INTERFACE I_Level EXTENDS I_Component

METHOD PUBLIC M_Attach : BOOL
VAR_INPUT
	iObject: 	I_Component;
END_VAR
END_METHOD

METHOD PUBLIC M_Detach : BOOL
VAR_INPUT
	iObject: 	I_Component;
END_VAR
END_METHOD

{attribute 'OPC.UA.DA.Property' := '1'}
{attribute 'monitoring' := 'call'}
PROPERTY PUBLIC P_Length : DINT
GET
END_GET
END_PROPERTY

END_INTERFACE

(* stored: Version 1.1.0.1
   Itf I_Level: Id {2fbecd23-39f8-0ccf-3cc5-99cfd7eae8ff}
   Method M_Attach: Id {61682764-95a3-005b-0687-ea823b4a0cdc}
   Method M_Detach: Id {fdfd1d32-8dea-096e-262a-fc1130b45f3b}
   Property P_Length: Id {8a2135b4-d434-0b40-34a8-c68dbf9ce1b5}
   Get Get: Id {66a86cd6-d653-0b3d-1595-194313d1aca7} *)
